VAR_GLOBAL
	{IF (defined (release))}
    	{attribute 'hide'}
	{END_IF}
	fbLogger:			FB_GlobalLogger;		// Global Logger, as default without module
	{attribute 'analysis' := '-33'}
	bSimulation:		BOOL;
END_VAR

(* stored: Version 1.1.0.1
   GVL Globals: Id {470c2b31-7e29-075f-0fd9-081ad8199996} *)
